TYPE UDT_HMI_LogItem :
STRUCT
	sTimestamp : STRING[23];
	sLevel : STRING;
	sMsg : T_MaxString;
	dColor_Bg : DWORD := E_Color.White; // Table row background color
END_STRUCT
END_TYPE

(* stored: Version 1.1.0.1, ProductVersion 3.1.4024.11
   DUT UDT_HMI_LogItem: Id {2d3e2c64-0033-40ec-a575-247769317aab} *)
